Staubli VAL3: init.pgx

public program init()
begin
  //Header begin
  //Description of program
  //  This program initializes the library's global variables.
  //  It has to be called once at the beginning of the users program
  //
  //History
  //  Creation : 16-04-08 - f.Rob
  //  KN: set quantity = 9 = max index of arrays (0-9)
  //Header end

  nNumberCylinder=nNumberCube=nNumberSphere=nNumberFrame=9
end
